Omron CX-Programmer project NewProject (CX-Programmer 9.51)

# PLC hydraulics_demo: CP1L M

## Program NewProgram1 (cyclic task 0)

### Section Section1

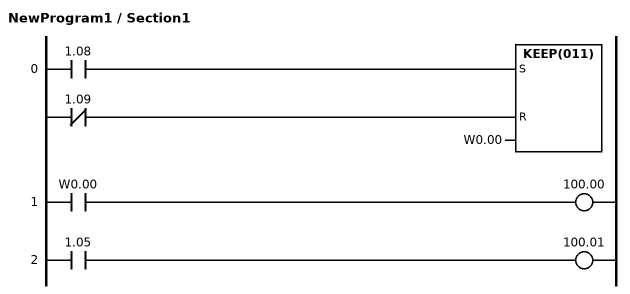
; rung 0
LD 1.08
LDNOT 1.09
KEEP(011) W0.00
; rung 1
LD W0.00
OUT 100.00
; rung 2
LD 1.05
OUT 100.01

### Section END
; rung 0
END(001)